(* CoDeSys 2.3 export: FB_WB_VALVE_LS.EXP *)

(* POU FB/FB_WB_VALVE_LS, ST *)
FUNCTION_BLOCK FB_WB_VALVE_LS
VAR_INPUT
	Enable : BOOL;
	Manual : BOOL;

	B_Open  : BOOL;
	B_Half  : BOOL;
	B_Close : BOOL;

	R_Open  : BOOL;
	R_Close : BOOL;

END_VAR
VAR_IN_OUT
	P   : ST_SENSOR_BAR;
	LS  : ST_SENSOR_POS;
	CFG : ST_WB_VALVE_LS_CFG;
END_VAR
VAR_OUTPUT
	OUT_Open  : BOOL;
	OUT_Close : BOOL;

	OUT_HP    : BYTE;
END_VAR
VAR
	State : WORD;

	IN_Hmi_Open  : BOOL;
	IN_Hmi_Close : BOOL;

	SI_Open  : FB_SMART_INPUT;
	SI_Half  : FB_SMART_INPUT;
	SI_Close : FB_SMART_INPUT;

	SI_Hmi_Open  : FB_SMART_INPUT;
	SI_Hmi_Close : FB_SMART_INPUT;
	SI_HmiR_Open  : FB_SMART_INPUT;
	SI_HmiR_Close : FB_SMART_INPUT;

	TimeCnt : REAL;
	TimeOut : BOOL;

	SF_Open : BOOL;
	SF_Half : BOOL;
	SF_Close : BOOL;

END_VAR
(*Check Inputs*)
SI_Open (In:= B_Open , T_Cont:= T#0ms, T_DClk:= T#0ms);
SI_Half (In:= B_Half , T_Cont:= T#0ms, T_DClk:= T#0ms);
SI_Close(In:= B_Close, T_Cont:= T#0ms, T_DClk:= T#0ms);

SI_Hmi_Open  (In:= IN_Hmi_Open , T_Cont:= T#0ms, T_DClk:= T#0ms);
SI_Hmi_Close (In:= IN_Hmi_Close, T_Cont:= T#0ms, T_DClk:= T#0ms);
SI_HmiR_Open (In:= R_Open , T_Cont:= T#0ms, T_DClk:= T#0ms);
SI_HmiR_Close(In:= R_Close, T_Cont:= T#0ms, T_DClk:= T#0ms);

SF_Open  := NOT LS.Err AND LS.Pos > 100.0 - CFG.LS_DB; 	(*OPEN  -> 100%*)
SF_Half  := NOT LS.Err AND LS.Pos > CFG.TgtLS_Half - CFG.LS_DB; (* CFG.LS_DB > ABS(CFG.TgtLS_Half - LS.Pos);*)
SF_Close := NOT LS.Err AND LS.Pos < CFG.LS_DB;  		(*CLOSE ->   0%*)

IF NOT Enable THEN
	OUT_Open  := FALSE;
	OUT_Close := FALSE;
	OUT_HP    := 0;

	TimeCnt := 0.0;
	State   := 0;
	RETURN;
END_IF

(*Check Time*)
TimeOut := TimeOut OR ( CFG.TimeMax > 0  AND TimeCnt > CFG.TimeMax );
TimeCnt := TimeCnt + CFG.Cycle;

(*Working States*)
CASE State OF

(*Init State*)
0:
	OUT_Open  := FALSE;
	OUT_Close := FALSE;
	OUT_HP    := 0;

	(*Manual*)
	IF Manual AND NOT P.AlMax THEN
		IF SI_Hmi_Open.Event = INIT_CONTINUOUS OR SI_HmiR_Open.Event = INIT_CONTINUOUS THEN
			OUT_Open  := TRUE;
			OUT_HP    := 1;
	
			TimeOut := FALSE; (*Reset TimeOut Error*)
			State   := 1001;  (*Next State*)

		ELSIF SI_Hmi_Close.Event = INIT_CONTINUOUS OR SI_HmiR_Close.Event = INIT_CONTINUOUS THEN
			OUT_Close := TRUE;
			OUT_HP    := 1;

			TimeOut := FALSE; (*Reset TimeOut Error*)
			State   := 1002;  (*Next State*)

		END_IF

	(*Automatico*)
	ELSIF NOT P.AlMax AND NOT LS.Err THEN
		IF SI_Open.Event = INIT_CONTINUOUS THEN
			OUT_Open  := TRUE;
			OUT_HP    := CFG.HP;

			TimeOut := FALSE; (*Reset TimeOut Error*)
			State   := 1010;  (*Next State*)

		ELSIF SI_Close.Event = INIT_CONTINUOUS THEN
			OUT_Close := TRUE;
			OUT_HP    := CFG.HP;

			TimeOut := FALSE; (*Reset TimeOut Error*)
			State   := 1020;  (*Next State*)

		ELSIF SI_Half.Event = INIT_CONTINUOUS THEN
			IF LS.Pos < CFG.TgtLS_Half - CFG.LS_DB THEN
				OUT_Open  := TRUE;
				OUT_HP    := CFG.HP;

				TimeOut := FALSE; (*Reset TimeOut Error*)
				State   := 1030;  (*Next State*)

			ELSIF LS.Pos > CFG.TgtLS_Half + CFG.LS_DB THEN
				OUT_Close := TRUE;
				OUT_HP    := CFG.HP;

				TimeOut := FALSE; (*Reset TimeOut Error*)
				State   := 1040;  (*Next State*)

			END_IF
		END_IF
	END_IF

    TimeCnt := 0.0; (*Time Count*)

(*Manual OPEN*)
1001:
	(*End*)
	IF SI_Hmi_Open.Event <> NONE OR SI_HmiR_Open.Event <> NONE
	OR SI_Hmi_Close.Event <> NONE OR SI_HmiR_Close.Event <> NONE
	OR TimeOut OR NOT Manual OR P.AlMax THEN
		OUT_Open  := FALSE;
		OUT_HP    := 0;
		State     := 0; (*Next State*)

	END_IF

(*Manual CLOSE*)
1002:
	(*End*)
	IF SI_Hmi_Open.Event <> NONE OR SI_HmiR_Open.Event <> NONE
	OR SI_Hmi_Close.Event <> NONE OR SI_HmiR_Close.Event <> NONE
	OR TimeOut OR NOT Manual OR P.AlMax THEN
		OUT_Close := FALSE;
		OUT_HP    := 0;
		State     := 0; (*Next State*)

	END_IF

(*Auto OPEN*)
1010,1030:
	(*End*)
	IF SI_Open.Event <> NONE OR SI_Half.Event <> NONE OR TimeOut OR Manual OR P.AlMax OR LS.Err THEN
		OUT_Open  := FALSE;
		OUT_HP    := 0;
		State     := 0; (*Next State*)

	ELSIF SI_Close.Event = INIT_CONTINUOUS THEN
		OUT_Open  := FALSE;
		OUT_Close := TRUE;
		State     := 1020; (*Next State*)

	ELSIF State = 1030 AND LS.Pos > CFG.TgtLS_Half - CFG.LS_DB THEN
		OUT_Open  := FALSE;
		OUT_HP    := 0;
		State     := 0; (*Next State*)

	ELSIF SF_Open THEN
		TimeCnt   := 0.0;
		State     := 1011; (*Next State*)

	END_IF

(*Push OPEN*)
1011:
	(*End*)
	IF SI_Open.Event <> NONE OR TimeOut OR TimeCnt > CFG.PushTime OR (CFG.PushP > 0 AND P.Bar > CFG.PushP) OR Manual OR P.AlMax THEN
		OUT_Open  := FALSE;
		OUT_HP    := 0;
		State     := 0; (*Next State*)

	ELSIF SI_Close.Event = INIT_CONTINUOUS THEN
		OUT_Open  := FALSE;
		OUT_Close := TRUE;
		State     := 1020; (*Next State*)

	END_IF

(*Auto CLOSE*)
1020,1040:
	(*End*)
	IF SI_Close.Event <> NONE OR SI_Half.Event <> NONE OR TimeOut OR Manual OR P.AlMax OR LS.Err THEN
		OUT_Close := FALSE;
		OUT_HP    := 0;
		State     := 0; (*Next State*)

	ELSIF SI_Open.Event = INIT_CONTINUOUS THEN
		OUT_Close := FALSE;
		OUT_Open  := TRUE;
		State     := 1010; (*Next State*)

	ELSIF State = 1040 AND LS.Pos < CFG.TgtLS_Half + CFG.LS_DB THEN
		OUT_Close := FALSE;
		OUT_HP    := 0;
		State     := 0; (*Next State*)

	ELSIF SF_Close THEN
		TimeCnt   := 0.0;
		State     := 1021; (*Next State*)

	END_IF

(*Push CLOSE*)
1021:
	(*End*)
	IF SI_Close.Event <> NONE OR TimeOut OR TimeCnt > CFG.PushTime OR (CFG.PushP > 0 AND P.Bar > CFG.PushP) OR Manual OR P.AlMax THEN
		OUT_Close := FALSE;
		OUT_HP    := 0;
		State     := 0; (*Next State*)

	ELSIF SI_Open.Event = INIT_CONTINUOUS THEN
		OUT_Close := FALSE;
		OUT_Open  := TRUE;
		State     := 1010; (*Next State*)

	END_IF


END_CASE
END_FUNCTION_BLOCK
